// TIA Portal V16 export
// export: Created 2021-11-12T13:31:01.9792213Z, ExportSetting WithDefaults, DisplayName Totally Integrated Automation Portal, DisplayVersion V16 Update 3, DisplayName TIA Portal Version Control Interface, DisplayVersion V16 Update 2, DisplayName TIA Portal Openness, DisplayVersion V16 Update 3, DisplayName SINAMICS Startdrive Advanced, DisplayVersion V16 Update 5, DisplayName SINAMICS Startdrive G130, G150, S120, S150, SINAMICS MV, S210, DisplayVersion V16 Update 5, DisplayName SINAMICS Startdrive G110M, G120, G120C, G120D, G120P, G115D, DisplayVersion V16 Update 5, DisplayName STEP 7 Professional, DisplayVersion V16 Update 3, DisplayName STEP 7 Safety, DisplayVersion V16, DisplayName WinCC UA Professional, DisplayVersion V16 Update 3
DATA_BLOCK "IDB_STD_System"   // DB2
{ DB_Accessible_From_OPC_UA := 'FALSE' }
VERSION : 0.1
// stored: AutoNumber false, DBAccessibleFromOPCUA false, InstanceOfName STD_System, InstanceOfType FB
"STD_System"
   // VAR
   //    SB1STDEdge_100ms : Bool;
   //    SB1STDEdge_200ms : Bool;
   //    SB1STDEdge_400ms : Bool;
   //    SB1STDEdge_500ms : Bool;
   //    SB1STDEdge_800ms : Bool;
   //    SB1STDEdge_1s : Bool;
   //    SB1STDEdge_1600ms : Bool;
   //    SB1STDEdge_2s : Bool;
   //    ST_TOFPulseEach10s { S7_SetPoint := 'True'} : TOF_TIME;
   //    ST_TOFPulseEach60s { S7_SetPoint := 'True'} : TOF_TIME;
   //    ST_TOFPulseEach600s { S7_SetPoint := 'True'} : TOF_TIME;
   //    ST_TOFPulseEach3600s { S7_SetPoint := 'True'} : TOF_TIME;
   //    ST_TONBlinking300ms { S7_SetPoint := 'True'} : TON_TIME;
   //    ST_TOFBlinking300ms { S7_SetPoint := 'True'} : TOF_TIME;
   //    ST_TONBlinking1sOn2sOff { S7_SetPoint := 'True'} : TON_TIME;
   //    ST_TOFBlinking1sOn2sOff { S7_SetPoint := 'True'} : TOF_TIME;
   //    ST_TOFDelayPulse500ms { S7_SetPoint := 'True'} : TOF_TIME;
   // END_VAR
BEGIN
END_DATA_BLOCK
